PROGRAM PRG_TEST
VAR
	HeatingCurve_Test : FC_HeatingCurve_Test;
	// FanControlTest : FB_FanControl_Test;
END_VAR

TcUnit.RUN();

END_PROGRAM

(* stored: Version 1.1.0.1, ProductVersion 3.1.4024.6
   POU PRG_TEST: Id {10f80d2f-bcd9-4294-9542-64c777584a32}, SpecialFunc None *)
